FUNCTION_BLOCK StartButton
VAR
	input AT %I* : BOOL;
END_VAR

PROPERTY IsPressed : BOOL
GET
IsPressed := input
END_GET
END_PROPERTY

PROPERTY IsReleased : BOOL
GET
IsReleased := NOT input;
END_GET
END_PROPERTY

END_FUNCTION_BLOCK

(* stored: Version 1.1.0.1, ProductVersion 3.1.4024.12
   POU StartButton: Id {dd361515-663c-4439-9f51-0e28f7d10fbb}, SpecialFunc None
   Property IsPressed: Id {ba4ac2d0-4cee-427f-832b-c659027bb1fc}
   Get Get: Id {87fc14ca-c9eb-42f8-b230-dd552e6bba8e}
   Property IsReleased: Id {7ded9d37-4e6b-4ad5-ab37-fcd95351a4ab}
   Get Get: Id {3d95c4d1-11fd-442c-99c3-518d80841ea8} *)
